FUNCTION_BLOCK PUBLIC ABSTRACT FB_PiezoDriveDS402 EXTENDS FB_PiezoDrive
VAR_INPUT
END_VAR
VAR_OUTPUT
END_VAR
VAR
    eInternalDriveState		: 	E_DS402_DRIVE_STATE;
	// reuse to absolute/relative moves
	eAxisState 				:  MC_AxisStates;
	rtReset					: R_TRIG;
	rtEnableDrive			: R_TRIG;
	rtDisbaleDrive			: F_TRIG;
	// Drive calibrated motion params
	nCalibratedVelocity			: DINT;
	nCalibratedAcceleration		: DINT;
	nCalibratedTargetPosition 	: DINT;
	
	fCalibratedActPos			: REAL;
	fCalibratedStoppedPos		: REAL;
	fOverride					: REAL;
	
	// axis status -- emulating some NC axis 
	bPowerEnabled		:  BOOL;
  	bOperational 		:  BOOL;
	PositiveDirection 	:  BOOL;
	NegativeDirection 	:  BOOL;
	NotMoving 			:  BOOL;
	NewTargetPosition 	:  BOOL;
	InPositionArea 		:  BOOL;
	InTargetPosition 	:  BOOL;
	StandStill 			:  BOOL;
	DiscreteMotion 		:  BOOL;
	ContinuousMotion 	:  BOOL;
	SynchronizedMotion 	:  BOOL;
 	ErrorStop 			:  BOOL;
 	Disabled 			:  BOOL;
 	Stopping 			:  BOOL;
	bHasJob 			:  BOOL;
    bMoveDone			:  BOOL;
	bMoveBusy			: BOOL;
END_VAR

METHOD Brake : BOOL
SUPER^.Brake();
END_METHOD

PROPERTY CalibratedAcceleration : DINT
GET
CalibratedAcceleration := nCalibratedAcceleration;
END_GET
END_PROPERTY

PROPERTY CalibratedActPos : REAL
GET
CalibratedActPos := fCalibratedActPos;
END_GET
END_PROPERTY

METHOD CalibratedMotionParams
VAR_INPUT
END_VAR
VAR

END_VAR
SUPER^.CalibratedMotionParams();
// Target Position
fCalibratedActPos :=  DINT_TO_REAL(SUPER^.stPiezoStage.nActualPosition) *  MAX(SUPER^.stPiezoStage.fscalingFactor, SUPER^.DefaultScalingFactor);
nCalibratedTargetPosition := LREAL_TO_DINT (SUPER^.stPiezoStage.fPosition / MAX(SUPER^.stPiezoStage.fscalingFactor, SUPER^.DefaultScalingFactor));
// set soft limit on drive params to avoid bumping hard on the end stops
nCalibratedVelocity := LIMIT(0, LREAL_TO_DINT (SUPER^.stPiezoStage.fVelocity / MAX(SUPER^.stPiezoStage.fscalingFactor, SUPER^.DefaultScalingFactor)), nCalibratedMaxVelocity);
nCalibratedAcceleration := LIMIT(0, LREAL_TO_DINT (SUPER^.stPiezoStage.fAcceleration / MAX(SUPER^.stPiezoStage.fscalingFactor, SUPER^.DefaultScalingFactor)), nCalibratedMaxAcceleration) ;
END_METHOD

PROPERTY CalibratedTargetPosition : DINT
GET
CalibratedTargetPosition:= nCalibratedTargetPosition;
END_GET
END_PROPERTY

PROPERTY CalibratedVelocity : DINT
GET
CalibratedVelocity := nCalibratedVelocity;
END_GET
END_PROPERTY

METHOD DS402StateMachine
VAR_INPUT
END_VAR
// Drive State Events and Operations
IF NOT __ISVALIDREF(SUPER^.stPiezoStage) THEN
    // we will return gracefully in the FAULT state
    ErrorMessage := 'FAULT: Drive interface not initialized';
    RETURN;
END_IF

(*switch on disable*)
IF NOT SUPER^.stPiezoStage.stPiezoDriveStatus.ReadyToSwitchOn
    AND NOT SUPER^.stPiezoStage.stPiezoDriveStatus.SwitchedOn
    AND NOT SUPER^.stPiezoStage.stPiezoDriveStatus.OperationEnabled
    AND NOT SUPER^.stPiezoStage.stPiezoDriveStatus.Fault
    AND  SUPER^.stPiezoStage.stPiezoDriveStatus.SwitchOnDisabled THEN
	
    eInternalDriveState  := E_DS402_DRIVE_STATE.SWITCH_ON_DISABLED;
END_IF

(*Ready to switch*)
IF  SUPER^.stPiezoStage.stPiezoDriveStatus.ReadyToSwitchOn
    AND NOT SUPER^.stPiezoStage.stPiezoDriveStatus.SwitchedOn
    AND NOT SUPER^.stPiezoStage.stPiezoDriveStatus.OperationEnabled
    AND NOT SUPER^.stPiezoStage.stPiezoDriveStatus.Fault
    AND SUPER^.stPiezoStage.stPiezoDriveStatus.QuickStopActive
    AND NOT SUPER^.stPiezoStage.stPiezoDriveStatus.SwitchOnDisabled THEN

    eInternalDriveState  := E_DS402_DRIVE_STATE.SWITCH_ON_READY;
END_IF

(*Switch on*)
IF  SUPER^.stPiezoStage.stPiezoDriveStatus.ReadyToSwitchOn
    AND SUPER^.stPiezoStage.stPiezoDriveStatus.SwitchedOn
    AND NOT SUPER^.stPiezoStage.stPiezoDriveStatus.OperationEnabled
    AND NOT SUPER^.stPiezoStage.stPiezoDriveStatus.Fault
    AND SUPER^.stPiezoStage.stPiezoDriveStatus.QuickStopActive
    AND NOT SUPER^.stPiezoStage.stPiezoDriveStatus.SwitchOnDisabled THEN

    eInternalDriveState  := E_DS402_DRIVE_STATE.SWITCH_ON;
END_IF

(*Operation enbaled*)
IF    SUPER^.stPiezoStage.stPiezoDriveStatus.ReadyToSwitchOn
    AND SUPER^.stPiezoStage.stPiezoDriveStatus.SwitchedOn
    AND SUPER^.stPiezoStage.stPiezoDriveStatus.OperationEnabled
    AND NOT SUPER^.stPiezoStage.stPiezoDriveStatus.Fault
    AND SUPER^.stPiezoStage.stPiezoDriveStatus.QuickStopActive
    AND NOT SUPER^.stPiezoStage.stPiezoDriveStatus.SwitchOnDisabled THEN

    eInternalDriveState  := E_DS402_DRIVE_STATE.OPERATION_ENABLED;
END_IF

(*Fault*)
IF  NOT  SUPER^.stPiezoStage.stPiezoDriveStatus.ReadyToSwitchOn
    AND NOT SUPER^.stPiezoStage.stPiezoDriveStatus.SwitchedOn
    AND NOT SUPER^.stPiezoStage.stPiezoDriveStatus.OperationEnabled
    AND SUPER^.stPiezoStage.stPiezoDriveStatus.Fault
    AND NOT SUPER^.stPiezoStage.stPiezoDriveStatus.SwitchOnDisabled THEN

    eInternalDriveState  := E_DS402_DRIVE_STATE.FAULT;
END_IF

(*Fault reaction active*)
IF    SUPER^.stPiezoStage.stPiezoDriveStatus.ReadyToSwitchOn
    AND SUPER^.stPiezoStage.stPiezoDriveStatus.SwitchedOn
    AND SUPER^.stPiezoStage.stPiezoDriveStatus.OperationEnabled
    AND SUPER^.stPiezoStage.stPiezoDriveStatus.Fault
    AND NOT SUPER^.stPiezoStage.stPiezoDriveStatus.SwitchOnDisabled THEN

    eInternalDriveState  := E_DS402_DRIVE_STATE.FAULT_ACTIVE;
END_IF

(*Quick Stop*)
IF    SUPER^.stPiezoStage.stPiezoDriveStatus.ReadyToSwitchOn
    AND SUPER^.stPiezoStage.stPiezoDriveStatus.SwitchedOn
    AND SUPER^.stPiezoStage.stPiezoDriveStatus.OperationEnabled
    AND NOT SUPER^.stPiezoStage.stPiezoDriveStatus.Fault
    AND SUPER^.stPiezoStage.stPiezoDriveStatus.VoltageEnabled
    AND NOT SUPER^.stPiezoStage.stPiezoDriveStatus.QuickStopActive
    AND NOT SUPER^.stPiezoStage.stPiezoDriveStatus.SwitchOnDisabled THEN

    eInternalDriveState  := E_DS402_DRIVE_STATE.QUICK_STOP_ACTIVE;
END_IF

CASE eInternalDriveState  OF

    E_DS402_DRIVE_STATE.SWITCH_ON_DISABLED:;
		// catch fault recovery here if needed

    E_DS402_DRIVE_STATE.SWITCH_ON_READY:;

    E_DS402_DRIVE_STATE.SWITCH_ON:;
		
    E_DS402_DRIVE_STATE.OPERATION_ENABLED:;
		bOperational := TRUE;

    E_DS402_DRIVE_STATE.FAULT:;
		// Theis is not a motion fault but rather hardware, lost of enabled wc or loss of calibration issue.
		// the same method we use to clear motion error too has the DS402 profil does not provide...
		THIS^.Reset();
		
    E_DS402_DRIVE_STATE.QUICK_STOP_ACTIVE:
		// return back to operation enabled: transition 16
		SUPER^.stPiezoStage.nPiezoDriveControl := 16#0F;

END_CASE

// Homing and absolute/relative moves only valid in this state
IF eInternalDriveState  <>  E_DS402_DRIVE_STATE.OPERATION_ENABLED THEN
		bOperational := FALSE;	
END_IF
END_METHOD

(*FB_Init is always available implicitly and it is used primarily for initialization.
The return value is not evaluated. For a specific influence, you can also declare the
methods explicitly and provide additional code there with the standard initialization
code. You can evaluate the return value.*)
METHOD FB_Init : BOOL
VAR_INPUT
    (* TRUE: the retain variables are initialized (reset warm / reset cold)*)
    bInitRetains	: BOOL;
    (* TRUE: the instance will be copied to the copy code afterward (online change)   *)
    bInCopyCode	: BOOL;
    stStage : REFERENCE TO  ST_PiezoStage;
END_VAR
//DS402Axis.stPiezoStageRef := stStage;
END_METHOD

METHOD Halt : BOOL
// Halt the move by setting bit 8 of the Control Word.
SUPER^.stPiezoStage.nPiezoDriveControl.8 := SUPER^.stPiezoStage.bHalt;
END_METHOD

METHOD Home : BOOL
SUPER^.Home();
END_METHOD

METHOD Interlock : BOOL
stPiezoStage.bLimitForwardEnable := (NOT SUPER^.stPiezoStage.stPiezoDriveStatus.InternalLimitActive);
stPiezoStage.bLimitBackwardEnable := (NOT SUPER^.stPiezoStage.stPiezoDriveStatus.InternalLimitActive);
// call common interlocks checker
SUPER^.Interlock();

// Handle auto-disable timing
bPrepareDisable S= stPiezoStage.nEnableMode = E_StageEnableMode.DURING_MOTION AND ftExec.Q;
// Delay the disable until we reach standstill, else brake issues or other race conditions
IF bPrepareDisable AND THIS^.eAxisState = MC_AXISSTATE_STANDSTILL THEN
    bPrepareDisable := FALSE;
    stPiezoStage.bEnable := FALSE;
END_IF

// Get a definitive bEnabled reading
CASE THIS^.eAxisState OF
    // We are not enabled if there is an issue
    MC_AXISSTATE_UNDEFINED, MC_AXISSTATE_DISABLED, MC_AXISSTATE_ERRORSTOP:
        SUPER^.stPiezoStage.bEnableDone := FALSE;
    ELSE
        SUPER^.stPiezoStage.bEnableDone := TRUE;
END_CASE

// IF doing profil positioning we should be able to do continous motion
// add an override here to account for it
IF stPiezoStage.stAxisStatus.bBusy AND NOT bExecute THEN
    // Wait for the previous move to end
    bExecute := FALSE;
	
ELSIF bMoveCmd THEN
    // Do not start the move until we have power and the safety system says it is OK
    bExecute := stPiezoStage.bExecute AND stPiezoStage.bAllEnable AND stPiezoStage.bEnableDone AND stPiezoStage.bSafetyReady;
ELSE
    bExecute := stPiezoStage.bExecute;
END_IF

// When we start, set the busy/done appropriately
rtExec(CLK:=bExecute);
IF rtExec.Q THEN
    SUPER^.stPiezoStage.bDone := FALSE;
END_IF

// definitive move cmds
bExecHome := bExecute AND stPiezoStage.nCommand = 10;
bExecMove := bExecute AND NOT bExecHome;
END_METHOD

METHOD Logger : BOOL
SUPER^.Logger();
END_METHOD

METHOD PUBLIC MoveAbsolute
END_METHOD

PROPERTY MoveBusy : BOOL
GET
MoveBusy := bHasJob;
END_GET
SET
bHasJob  := MoveBusy;
END_SET
END_PROPERTY

PROPERTY MoveDone : BOOL
GET
MoveDone := bMoveDone;
END_GET
SET
bMoveDone := MoveDone;
END_SET
END_PROPERTY

METHOD MoveRelative
VAR_INPUT
END_VAR
END_METHOD

METHOD PUBLIC ABSTRACT MoveVelocity
END_METHOD

METHOD Power : BOOL
rtEnableDrive(CLK:=SUPER^.stPiezoStage.bAllEnable);
rtDisbaleDrive(CLK:=SUPER^.stPiezoStage.bAllEnable);

// Enabled the drive: the client code must wait for state transitions.
IF rtEnableDrive.Q THEN
	// Voltage on, close loop operations
	SUPER^.stPiezoStage.nPiezoDriveControl := 16#0F;
	fOverride := 100.0;
END_IF

IF rtDisbaleDrive.Q THEN
	fOverride := 0.0;
END_IF
END_METHOD

METHOD ReadStatus
VAR_INPUT
END_VAR
END_METHOD

METHOD Reset : BOOL
// Try to clear any faults if they are present by setting bit 7 of the Control Word.
rtReset(CLK:=SUPER^.stPiezoStage.bReset);
IF rtReset.Q THEN
	SUPER^.stPiezoStage.nPiezoDriveControl := 16#80;
	// Reset everything when bReset is flagged
    SUPER^.stPiezoStage.bEnable := FALSE;
    SUPER^.stPiezoStage.bReset := FALSE;
    SUPER^.stPiezoStage.bExecute := FALSE;
    SUPER^.stPiezoStage.bError := FALSE;
    SUPER^.stPiezoStage.nErrorId := 0;
    SUPER^.stPiezoStage.sErrorMessage := '';
    SUPER^.stPiezoStage.sCustomErrorMessage := '';
    SUPER^.bExecute := FALSE;
END_IF
END_METHOD

METHOD SyncEpicsStatus
VAR_INPUT
END_VAR
//Status struct for EPICS communication
SUPER^.stPiezoStage.stAxisStatus.bEnable:=SUPER^.stPiezoStage.bAllEnable;
SUPER^.stPiezoStage.stAxisStatus.bEnabled:=SUPER^.stPiezoStage.bEnableDone; // account for PowerEnable from power block
SUPER^.stPiezoStage.stAxisStatus.bError:=SUPER^.stPiezoStage.bError;
SUPER^.stPiezoStage.stAxisStatus.bExecute:=SUPER^.stPiezoStage.bExecute;
SUPER^.stPiezoStage.stAxisStatus.bHomeSensor:=SUPER^.stPiezoStage.bHome;
SUPER^.stPiezoStage.stAxisStatus.bLimitBwd:=SUPER^.stPiezoStage.bAllBackwardEnable;
SUPER^.stPiezoStage.stAxisStatus.bLimitFwd:=SUPER^.stPiezoStage.bAllForwardEnable;
SUPER^.stPiezoStage.stAxisStatus.bReset:=SUPER^.stPiezoStage.bReset;
SUPER^.stPiezoStage.stAxisStatus.fAcceleration:=SUPER^.stPiezoStage.fAcceleration;
SUPER^.stPiezoStage.stAxisStatus.fActDiff:=SUPER^.stPiezoStage.fPosDiff;
SUPER^.stPiezoStage.stAxisStatus.fActPosition:=THIS^.CalibratedActPos;
SUPER^.stPiezoStage.stAxisStatus.fActVelocity:=SUPER^.stPiezoStage.fVelocity;
SUPER^.stPiezoStage.stAxisStatus.fDeceleration:=SUPER^.stPiezoStage.fAcceleration;
SUPER^.stPiezoStage.stAxisStatus.fOverride:=THIS^.fOverride;
SUPER^.stPiezoStage.stAxisStatus.fPosition:=SUPER^.stPiezoStage.fPosition;
SUPER^.stPiezoStage.stAxisStatus.fVelocity:=SUPER^.stPiezoStage.fVelocity;
SUPER^.stPiezoStage.stAxisStatus.nCmdData:=SUPER^.stPiezoStage.nCmdData;  //Or nCmdDataLocal
SUPER^.stPiezoStage.stAxisStatus.nCommand:=SUPER^.stPiezoStage.nCommand;  //Or nCommandLocal
SUPER^.stPiezoStage.stAxisStatus.nErrorId:=SUPER^.stPiezoStage.nErrorId;
SUPER^.stPiezoStage.stAxisStatus.bBusy:=SUPER^.stPiezoStage.bBusy;
SUPER^.stPiezoStage.stAxisStatus.bHomed:=SUPER^.stPiezoStage.bHomed;
END_METHOD

END_FUNCTION_BLOCK

(* stored: Version 1.1.0.1
   POU FB_PiezoDriveDS402: Id {767dade8-900b-419e-8640-c738938dffde}, SpecialFunc None
   Method Brake: Id {e5829bdb-4f85-41d9-84ca-59543bab5ffb}
   Property CalibratedAcceleration: Id {c9db77b1-cfd0-4d09-b550-344bf9246222}
   Get Get: Id {0de4f123-8d8a-4161-9634-33cbec6d4458}
   Property CalibratedActPos: Id {f59b6d0c-3ed5-49c8-8c42-f3fe81b218e0}
   Get Get: Id {7008e174-6003-4a34-8527-bc95fa10dfd5}
   Method CalibratedMotionParams: Id {ac17b7c4-a540-4db8-be71-88c2b2fc9fb9}
   Property CalibratedTargetPosition: Id {81813abc-be79-4b01-bd0b-013ad1ba8c86}
   Get Get: Id {b29f2fdd-a221-4a00-b566-55ff2dd3354a}
   Property CalibratedVelocity: Id {54e27d08-db1c-4a56-8d6f-ee25264ddf78}
   Get Get: Id {55f6b951-9e85-4976-9d4e-affbfb1a904d}
   Method DS402StateMachine: Id {d963b9d7-d9e1-4a33-bb79-0f8a7e20b1de}
   Method FB_Init: Id {8fccdb5f-b457-4637-ae44-ff5efe2142a7}
   Method Halt: Id {7f626c89-4c25-446a-aadf-2d7158be6cb2}
   Method Home: Id {d33ee575-f547-404d-bc45-25b73c38be5a}
   Method Interlock: Id {36207be0-7a17-466d-9c72-e0f495170f07}
   Method Logger: Id {c74ad8cb-1745-4df8-b83c-c7761caffd8e}
   Method MoveAbsolute: Id {8f7c0eeb-20cc-4e52-be08-683acc155eb8}
   Property MoveBusy: Id {d58c53d5-d71e-4dfb-81d9-c7fda2274825}
   Get Get: Id {0dc6e9a0-7a00-4339-8717-53ef63ce7bac}
   Set Set: Id {2b796103-4887-45ce-b787-f19ffce80544}
   Property MoveDone: Id {4dfc439a-a1c1-4c95-b749-95d177fa4901}
   Get Get: Id {8556348b-daa4-4c56-8993-087102c74a94}
   Set Set: Id {16c38ccc-bd1b-40f2-bbe5-f6aaca214440}
   Method MoveRelative: Id {274dd405-a068-4680-bb9e-fe5025f2f908}
   Method MoveVelocity: Id {1b2e41e2-09a4-4d38-9d3b-52ed665fafd3}
   Method Power: Id {634342db-4980-4103-96da-256cbacd69e1}
   Method ReadStatus: Id {222b82c3-b7d6-4787-9577-5abf84745d3e}
   Method Reset: Id {ca77c887-2b90-4375-866f-a9f6ff5b335c}
   Method SyncEpicsStatus: Id {0ec1ab11-3e34-4193-8590-6aaa07110b4c} *)
